{attribute 'linkalways'} 
{attribute 'no_explicit_call' := 'This FB is a CLASS and must be accessed using methods or properties'}
{attribute 'enable_dynamic_creation'}
FUNCTION_BLOCK _ETcVnStructuringElementShape EXTENDS EnumDatatypeBase
VAR
	localData : ETcVnStructuringElementShape;
	activeData : REFERENCE TO ETcVnStructuringElementShape;
	enumBaseDatatype : _DINT(localData);
END_VAR

METHOD PRIVATE AddLocalEnumeration
VAR_INPUT
	Enumeration : T_MAXSTRING;
	Value : ETcVnStructuringElementShape;
END_VAR
AddEnumeration(Enumeration, Value);
END_METHOD

PROPERTY PUBLIC Address : PVOID
GET
Address := ADR(activeData);
END_GET
END_PROPERTY

METHOD PUBLIC ClearReference
VAR_INPUT
END_VAR
activeData REF= localData;
SetBaseDatatypeReference();
END_METHOD

METHOD PUBLIC Clone : I_Datatype
VAR
    pClone : POINTER TO _ETcVnStructuringElementShape;
END_VAR
pClone := __NEW(_ETcVnStructuringElementShape(InitialValue := Value));
Clone := pClone^;
END_METHOD

METHOD FB_init : BOOL
VAR_INPUT
	bInitRetains : BOOL; // if TRUE, the retain variables are initialized (warm start / cold start)
	bInCopyCode : BOOL;  // if TRUE, the instance afterwards gets moved into the copy code (online change)
	InitialValue : ETcVnStructuringElementShape;
END_VAR
localData := InitialValue;
AddBaseDatatype(enumBaseDatatype);
ClearReference();

AddLocalEnumeration('TCVN_SES_RECTANGLE', ETcVnStructuringElementShape.TCVN_SES_RECTANGLE);
AddLocalEnumeration('TCVN_SES_CROSS', ETcVnStructuringElementShape.TCVN_SES_CROSS);
AddLocalEnumeration('TCVN_SES_ELLIPSE', ETcVnStructuringElementShape.TCVN_SES_ELLIPSE);
END_METHOD

PROPERTY PUBLIC Identifier : T_MAXSTRING
GET
Identifier := 'ETcVnStructuringElementShape';
END_GET
END_PROPERTY

METHOD IsEnumeratorValueEqual : BOOL
VAR_INPUT
	Enumerator : I_KeyValueForwardEnumerator;
END_VAR
VAR
	storedValue : ETcVnStructuringElementShape;
END_VAR
IF NOT Enumerator.TryGet(storedValue) THEN
	RETURN;
END_IF

IsEnumeratorValueEqual := storedValue = activeData;
END_METHOD

METHOD PUBLIC MakeReferenceTo
VAR_INPUT
	ReferenceTarget : REFERENCE TO ETcVnStructuringElementShape;
END_VAR
activeData REF= ReferenceTarget;
SetBaseDatatypeReference();
END_METHOD

METHOD PROTECTED SetBaseDatatypeReference
VAR_INPUT
END_VAR
enumBaseDatatype.MakeReferenceTo(activeData);
END_METHOD

PROPERTY PUBLIC Size : UDINT
GET
Size := SIZEOF(activeData);
END_GET
END_PROPERTY

METHOD TryMakeReferenceTo : BOOL
VAR_INPUT
	Target : I_Datatype;
END_VAR
VAR
	pTargetData : POINTER TO ETcVnStructuringElementShape;
END_VAR
IF NOT IsEquivalentTo(Target) THEN
	RETURN;
END_IF

pTargetData := Target.Address;
activeData REF= pTargetData^;
SetBaseDatatypeReference();
TryMakeReferenceTo := TRUE;
END_METHOD

PROPERTY PUBLIC Value : ETcVnStructuringElementShape
GET
Value := activeData;
END_GET
SET
activeData := Value;
END_SET
END_PROPERTY

END_FUNCTION_BLOCK

(* stored: Version 1.1.0.1, ProductVersion 3.1.4024.13
   POU _ETcVnStructuringElementShape: Id {98728f69-0608-0d2b-10b0-74611e94f838}, SpecialFunc None
   Folder Core: Id {139c0530-d3e0-0fbd-0676-4f5af5f1346a}
   Folder Protected: Id {05a377e6-2fd2-035a-3b3f-f326f30aaebe}
   Folder Customize: Id {6ee64d37-e9c5-0bfd-0409-d5bf2864dd69}
   Folder Constructor: Id {b1c8afc6-282a-0502-215b-d81ce3079bd8}
   Folder Private: Id {cb20952e-2cdf-0515-2b56-db8d43aa7dea}
   Folder Protected: Id {d4b3f6cc-e452-0aad-1187-e9dabdee7998}
   Method AddLocalEnumeration: Id {5c0beae6-790d-0715-1fbc-e987da497e9f}
   Property Address: Id {6e250ae5-1206-0085-13e4-6e12da955200}
   Get Get: Id {e12e85c3-b5ae-02cc-148b-a7d6239f65c5}
   Method ClearReference: Id {223b2dbc-b101-0810-2e82-54e043b8eaf7}
   Method Clone: Id {7f29dc26-3af6-0c8d-06c1-be66f7382347}
   Method FB_init: Id {26b61613-c7e1-0a0b-0ea4-aab97e68ca7b}
   Property Identifier: Id {1c4a4fd8-d362-02f8-3be8-c8bdf926fddb}
   Get Get: Id {71467f8e-8dd6-0ce5-3345-12339c5cbe75}
   Method IsEnumeratorValueEqual: Id {a3a3020d-5216-044e-15ca-119adee6a51d}
   Method MakeReferenceTo: Id {52082723-81d8-07b5-27fd-305501175631}
   Method SetBaseDatatypeReference: Id {74950eb2-56c1-0559-1cfe-5f7817c8066b}
   Property Size: Id {7128782b-a464-0384-3872-72652d5866f1}
   Get Get: Id {051af4df-bfd3-0e38-1b56-932a7634532e}
   Method TryMakeReferenceTo: Id {722d836a-9c9a-087b-0562-d8772856cecb}
   Property Value: Id {812f6903-e6a4-0b4f-17a3-d7683961751f}
   Get Get: Id {7bcfe54d-991d-0b1b-0158-c526ef4f0857}
   Set Set: Id {511a79fe-34cc-0abb-1a51-057fd8b724bd} *)
